TYPE E_GS1_CodeLvl :
(
	E_LVL_NONE,
	E_LEVEL1,
	E_LEVEL2,
	E_LEVEL3
);
END_TYPE

(* stored: Version 1.1.0.1
   DUT E_GS1_CodeLvl: Id {45e9d865-8f42-4866-bc57-0da22526558a} *)
